// TIA Portal V17 export
// export: Created 2025-04-09T08:02:53.4997425Z, ExportSetting WithDefaults, DisplayName Totally Integrated Automation Portal, DisplayVersion V17 Update 8, DisplayName TIA Portal Openness, DisplayVersion V17 Update 8, DisplayName TIA Portal Version Control Interface, DisplayVersion V17, DisplayName SINAMICS Startdrive Advanced, DisplayVersion V17 SP2, DisplayName SINAMICS Startdrive G110M, G120, G120C, G120D, G120P, G115D, DisplayVersion V17 SP2, DisplayName SINAMICS Startdrive G130, G150, S120, S150, SINAMICS MV, S210, DisplayVersion V17 SP2, DisplayName STEP 7 Professional, DisplayVersion V17 Update 8, DisplayName SINUMERIK ONE STEP 7 Toolbox, DisplayVersion V17 Update 12, DisplayName SINUMERIK ONE PLC Basic Program Plus, DisplayVersion V17 Update 12, DisplayName SINUMERIK 840D sl STEP 7 Toolbox, DisplayVersion V17 Update 12, DisplayName STEP 7 Safety, DisplayVersion V17 Update 6, DisplayName WinCC Advanced, DisplayVersion V17 Update 8
FUNCTION "FC7000_SAFETY_DOORS" : Void   // FC7000, LAD
{ S7_Optimized_Access := 'FALSE' }
AUTHOR : ETXETAR
VERSION : 1.0
// stored: AutoNumber false, IsIECCheckEnabled false, SetENOAutomatically false, UDAEnableTagReadback false
BEGIN

REGION Network 1: CALL FC7002 UNIT 01 STATION 2 SAFETY DOOR
   // 2#0000_0001 OPTIONS 0 BIT 0 IMMEDIATE STOP REACTION OPTION
   // 2#0000_0010 OPTIONS 0 BIT 1 SEOC WARNING REACTION OPTION
   // 2#0000_0100 OPTIONS 0 BIT 2 CLOSED SENSOR INPUT OPTION
   // 2#0000_1000 OPTIONS 0 BIT 3 CIRCUIT E2 OPTION
   // 2#0001_0000 OPTIONS 0 BIT 4 PNEUMATIC DRIVE OPTION
   // 2#0010_0000 OPTIONS 0 BIT 5 GANTRY ROBOT OK TO OPEN OPTION
   // 2#0100_0000 OPTIONS 0 BIT 6 SPARE OPTION
   // 2#1000_0000 OPTIONS 0 BIT 7 SPARE OPTION
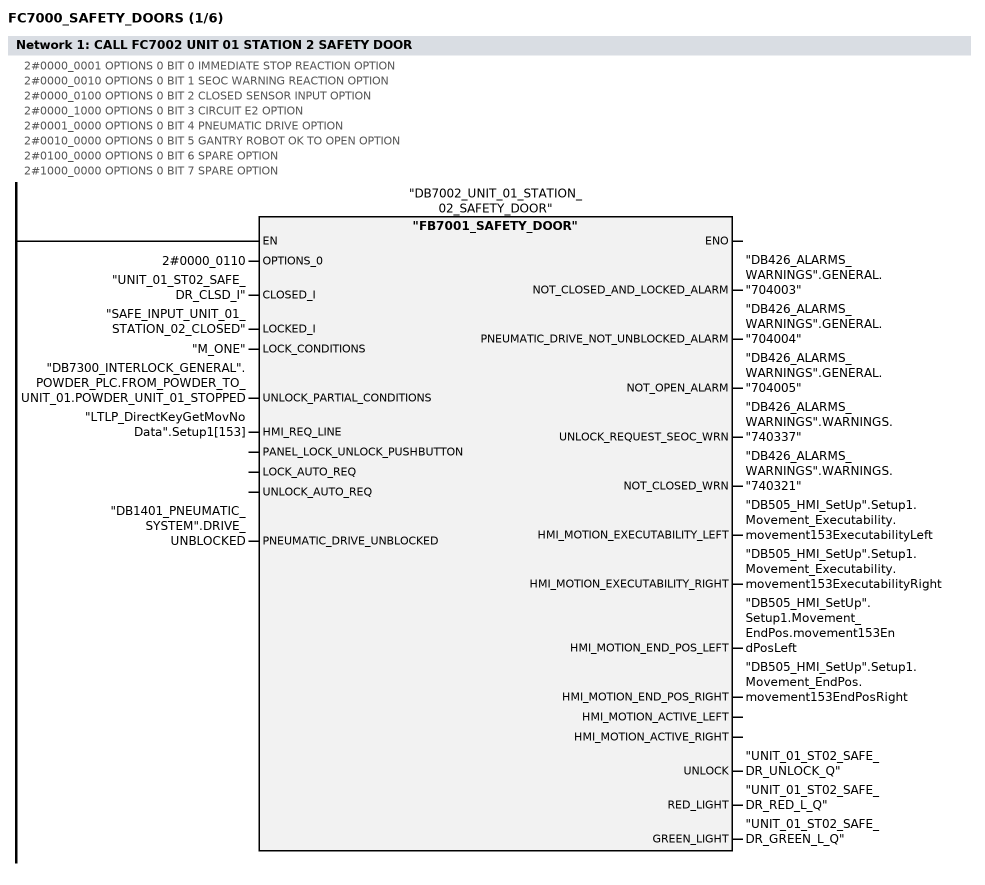
   RUNG wire#powerrail
      "DB7002_UNIT_01_STATION_02_SAFETY_DOOR"(OPTIONS_0 := 2#0000_0110, CLOSED_I := "UNIT_01_ST02_SAFE_DR_CLSD_I", LOCKED_I := "SAFE_INPUT_UNIT_01_STATION_02_CLOSED", LOCK_CONDITIONS := "M_ONE", UNLOCK_PARTIAL_CONDITIONS := "DB7300_INTERLOCK_GENERAL".POWDER_PLC.FROM_POWDER_TO_UNIT_01.POWDER_UNIT_01_STOPPED, HMI_REQ_LINE := "LTLP_DirectKeyGetMovNoData".Setup1[153], PANEL_LOCK_UNLOCK_PUSHBUTTON :=, LOCK_AUTO_REQ :=, UNLOCK_AUTO_REQ :=, PNEUMATIC_DRIVE_UNBLOCKED := "DB1401_PNEUMATIC_SYSTEM".DRIVE_UNBLOCKED, NOT_CLOSED_AND_LOCKED_ALARM => "DB426_ALARMS_WARNINGS".GENERAL."704003", PNEUMATIC_DRIVE_NOT_UNBLOCKED_ALARM => "DB426_ALARMS_WARNINGS".GENERAL."704004", NOT_OPEN_ALARM => "DB426_ALARMS_WARNINGS".GENERAL."704005", UNLOCK_REQUEST_SEOC_WRN => "DB426_ALARMS_WARNINGS".WARNINGS."740337", NOT_CLOSED_WRN => "DB426_ALARMS_WARNINGS".WARNINGS."740321", HMI_MOTION_EXECUTABILITY_LEFT => "DB505_HMI_SetUp".Setup1.Movement_Executability.movement153ExecutabilityLeft, HMI_MOTION_EXECUTABILITY_RIGHT => "DB505_HMI_SetUp".Setup1.Movement_Executability.movement153ExecutabilityRight, HMI_MOTION_END_POS_LEFT => "DB505_HMI_SetUp".Setup1.Movement_EndPos.movement153EndPosLeft, HMI_MOTION_END_POS_RIGHT => "DB505_HMI_SetUp".Setup1.Movement_EndPos.movement153EndPosRight, HMI_MOTION_ACTIVE_LEFT =>, HMI_MOTION_ACTIVE_RIGHT =>, UNLOCK => "UNIT_01_ST02_SAFE_DR_UNLOCK_Q", RED_LIGHT => "UNIT_01_ST02_SAFE_DR_RED_L_Q", GREEN_LIGHT => "UNIT_01_ST02_SAFE_DR_GREEN_L_Q")
   END_RUNG
   // the same network as SCL:
   "DB7002_UNIT_01_STATION_02_SAFETY_DOOR"(OPTIONS_0 := 2#0000_0110,   // "FB7001_SAFETY_DOOR"
                           CLOSED_I := "UNIT_01_ST02_SAFE_DR_CLSD_I",
                           LOCKED_I := "SAFE_INPUT_UNIT_01_STATION_02_CLOSED",
                           LOCK_CONDITIONS := "M_ONE",
                           UNLOCK_PARTIAL_CONDITIONS := "DB7300_INTERLOCK_GENERAL".POWDER_PLC.FROM_POWDER_TO_UNIT_01.POWDER_UNIT_01_STOPPED,
                           HMI_REQ_LINE := "LTLP_DirectKeyGetMovNoData".Setup1[153],
                           PNEUMATIC_DRIVE_UNBLOCKED := "DB1401_PNEUMATIC_SYSTEM".DRIVE_UNBLOCKED,
                           NOT_CLOSED_AND_LOCKED_ALARM => "DB426_ALARMS_WARNINGS".GENERAL."704003",
                           PNEUMATIC_DRIVE_NOT_UNBLOCKED_ALARM => "DB426_ALARMS_WARNINGS".GENERAL."704004",
                           NOT_OPEN_ALARM => "DB426_ALARMS_WARNINGS".GENERAL."704005",
                           UNLOCK_REQUEST_SEOC_WRN => "DB426_ALARMS_WARNINGS".WARNINGS."740337",
                           NOT_CLOSED_WRN => "DB426_ALARMS_WARNINGS".WARNINGS."740321",
                           HMI_MOTION_EXECUTABILITY_LEFT => "DB505_HMI_SetUp".Setup1.Movement_Executability.movement153ExecutabilityLeft,
                           HMI_MOTION_EXECUTABILITY_RIGHT => "DB505_HMI_SetUp".Setup1.Movement_Executability.movement153ExecutabilityRight,
                           HMI_MOTION_END_POS_LEFT => "DB505_HMI_SetUp".Setup1.Movement_EndPos.movement153EndPosLeft,
                           HMI_MOTION_END_POS_RIGHT => "DB505_HMI_SetUp".Setup1.Movement_EndPos.movement153EndPosRight,
                           UNLOCK => "UNIT_01_ST02_SAFE_DR_UNLOCK_Q",
                           RED_LIGHT => "UNIT_01_ST02_SAFE_DR_RED_L_Q",
                           GREEN_LIGHT => "UNIT_01_ST02_SAFE_DR_GREEN_L_Q");
END_REGION

REGION Network 2: CALL FC7002 UNIT 01 STATION 4 SAFETY DOOR
   // 2#0000_0001 OPTIONS 0 BIT 0 IMMEDIATE STOP REACTION OPTION
   // 2#0000_0010 OPTIONS 0 BIT 1 SEOC WARNING REACTION OPTION
   // 2#0000_0100 OPTIONS 0 BIT 2 CLOSED SENSOR INPUT OPTION
   // 2#0000_1000 OPTIONS 0 BIT 3 CIRCUIT E2 OPTION
   // 2#0001_0000 OPTIONS 0 BIT 4 PNEUMATIC DRIVE OPTION
   // 2#0010_0000 OPTIONS 0 BIT 5 GANTRY ROBOT OK TO OPEN OPTION
   // 2#0100_0000 OPTIONS 0 BIT 6 SPARE OPTION
   // 2#1000_0000 OPTIONS 0 BIT 7 SPARE OPTION
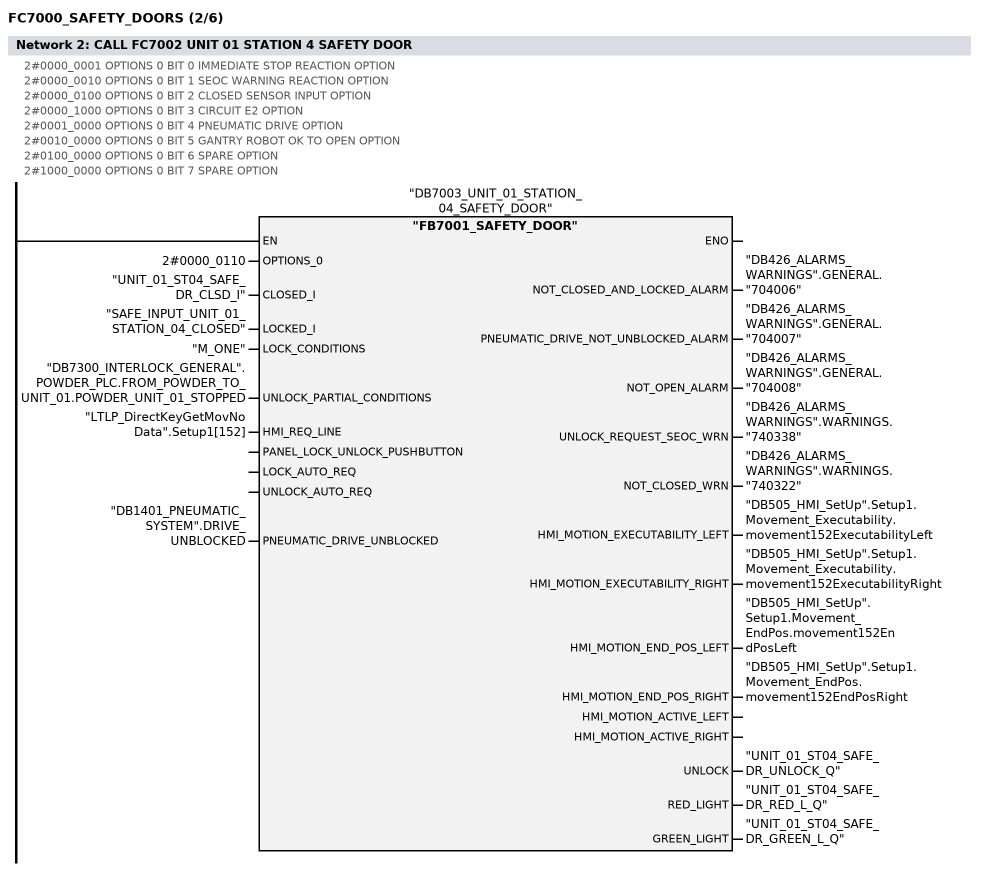
   RUNG wire#powerrail
      "DB7003_UNIT_01_STATION_04_SAFETY_DOOR"(OPTIONS_0 := 2#0000_0110, CLOSED_I := "UNIT_01_ST04_SAFE_DR_CLSD_I", LOCKED_I := "SAFE_INPUT_UNIT_01_STATION_04_CLOSED", LOCK_CONDITIONS := "M_ONE", UNLOCK_PARTIAL_CONDITIONS := "DB7300_INTERLOCK_GENERAL".POWDER_PLC.FROM_POWDER_TO_UNIT_01.POWDER_UNIT_01_STOPPED, HMI_REQ_LINE := "LTLP_DirectKeyGetMovNoData".Setup1[152], PANEL_LOCK_UNLOCK_PUSHBUTTON :=, LOCK_AUTO_REQ :=, UNLOCK_AUTO_REQ :=, PNEUMATIC_DRIVE_UNBLOCKED := "DB1401_PNEUMATIC_SYSTEM".DRIVE_UNBLOCKED, NOT_CLOSED_AND_LOCKED_ALARM => "DB426_ALARMS_WARNINGS".GENERAL."704006", PNEUMATIC_DRIVE_NOT_UNBLOCKED_ALARM => "DB426_ALARMS_WARNINGS".GENERAL."704007", NOT_OPEN_ALARM => "DB426_ALARMS_WARNINGS".GENERAL."704008", UNLOCK_REQUEST_SEOC_WRN => "DB426_ALARMS_WARNINGS".WARNINGS."740338", NOT_CLOSED_WRN => "DB426_ALARMS_WARNINGS".WARNINGS."740322", HMI_MOTION_EXECUTABILITY_LEFT => "DB505_HMI_SetUp".Setup1.Movement_Executability.movement152ExecutabilityLeft, HMI_MOTION_EXECUTABILITY_RIGHT => "DB505_HMI_SetUp".Setup1.Movement_Executability.movement152ExecutabilityRight, HMI_MOTION_END_POS_LEFT => "DB505_HMI_SetUp".Setup1.Movement_EndPos.movement152EndPosLeft, HMI_MOTION_END_POS_RIGHT => "DB505_HMI_SetUp".Setup1.Movement_EndPos.movement152EndPosRight, HMI_MOTION_ACTIVE_LEFT =>, HMI_MOTION_ACTIVE_RIGHT =>, UNLOCK => "UNIT_01_ST04_SAFE_DR_UNLOCK_Q", RED_LIGHT => "UNIT_01_ST04_SAFE_DR_RED_L_Q", GREEN_LIGHT => "UNIT_01_ST04_SAFE_DR_GREEN_L_Q")
   END_RUNG
   // the same network as SCL:
   "DB7003_UNIT_01_STATION_04_SAFETY_DOOR"(OPTIONS_0 := 2#0000_0110,   // "FB7001_SAFETY_DOOR"
                           CLOSED_I := "UNIT_01_ST04_SAFE_DR_CLSD_I",
                           LOCKED_I := "SAFE_INPUT_UNIT_01_STATION_04_CLOSED",
                           LOCK_CONDITIONS := "M_ONE",
                           UNLOCK_PARTIAL_CONDITIONS := "DB7300_INTERLOCK_GENERAL".POWDER_PLC.FROM_POWDER_TO_UNIT_01.POWDER_UNIT_01_STOPPED,
                           HMI_REQ_LINE := "LTLP_DirectKeyGetMovNoData".Setup1[152],
                           PNEUMATIC_DRIVE_UNBLOCKED := "DB1401_PNEUMATIC_SYSTEM".DRIVE_UNBLOCKED,
                           NOT_CLOSED_AND_LOCKED_ALARM => "DB426_ALARMS_WARNINGS".GENERAL."704006",
                           PNEUMATIC_DRIVE_NOT_UNBLOCKED_ALARM => "DB426_ALARMS_WARNINGS".GENERAL."704007",
                           NOT_OPEN_ALARM => "DB426_ALARMS_WARNINGS".GENERAL."704008",
                           UNLOCK_REQUEST_SEOC_WRN => "DB426_ALARMS_WARNINGS".WARNINGS."740338",
                           NOT_CLOSED_WRN => "DB426_ALARMS_WARNINGS".WARNINGS."740322",
                           HMI_MOTION_EXECUTABILITY_LEFT => "DB505_HMI_SetUp".Setup1.Movement_Executability.movement152ExecutabilityLeft,
                           HMI_MOTION_EXECUTABILITY_RIGHT => "DB505_HMI_SetUp".Setup1.Movement_Executability.movement152ExecutabilityRight,
                           HMI_MOTION_END_POS_LEFT => "DB505_HMI_SetUp".Setup1.Movement_EndPos.movement152EndPosLeft,
                           HMI_MOTION_END_POS_RIGHT => "DB505_HMI_SetUp".Setup1.Movement_EndPos.movement152EndPosRight,
                           UNLOCK => "UNIT_01_ST04_SAFE_DR_UNLOCK_Q",
                           RED_LIGHT => "UNIT_01_ST04_SAFE_DR_RED_L_Q",
                           GREEN_LIGHT => "UNIT_01_ST04_SAFE_DR_GREEN_L_Q");
END_REGION

REGION Network 3: CALL FC7001 UNIT 01 MAIN SAFETY DOOR
   // 2#0000_0001 OPTIONS 0 BIT 0 IMMEDIATE STOP REACTION OPTION
   // 2#0000_0010 OPTIONS 0 BIT 1 SEOC WARNING REACTION OPTION
   // 2#0000_0100 OPTIONS 0 BIT 2 CLOSED SENSOR INPUT OPTION
   // 2#0000_1000 OPTIONS 0 BIT 3 CIRCUIT E2 OPTION
   // 2#0001_0000 OPTIONS 0 BIT 4 PNEUMATIC DRIVE OPTION
   // 2#0010_0000 OPTIONS 0 BIT 5 GANTRY ROBOT OK TO OPEN OPTION
   // 2#0100_0000 OPTIONS 0 BIT 6 SPARE OPTION
   // 2#1000_0000 OPTIONS 0 BIT 7 SPARE OPTION
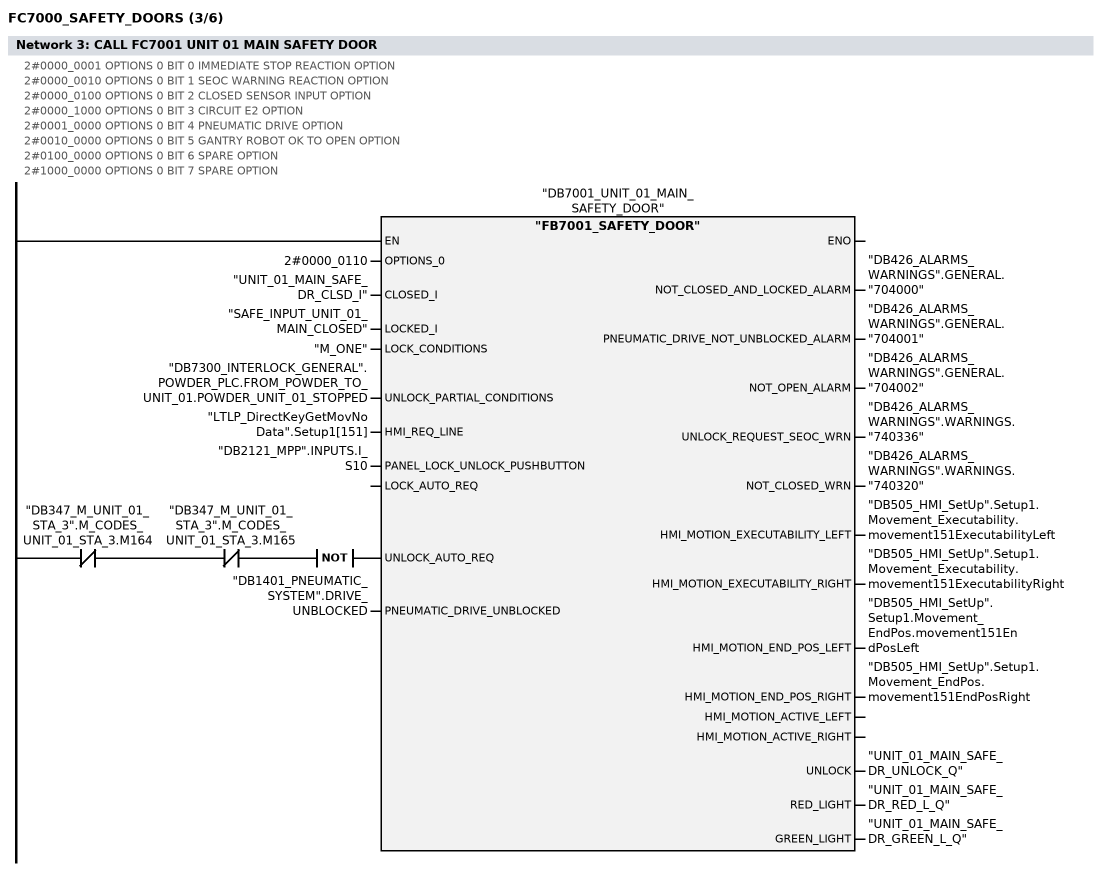
   RUNG wire#powerrail
      "DB7001_UNIT_01_MAIN_SAFETY_DOOR"(UNLOCK_AUTO_REQ := wire#w1, OPTIONS_0 := 2#0000_0110, CLOSED_I := "UNIT_01_MAIN_SAFE_DR_CLSD_I", LOCKED_I := "SAFE_INPUT_UNIT_01_MAIN_CLOSED", LOCK_CONDITIONS := "M_ONE", UNLOCK_PARTIAL_CONDITIONS := "DB7300_INTERLOCK_GENERAL".POWDER_PLC.FROM_POWDER_TO_UNIT_01.POWDER_UNIT_01_STOPPED, HMI_REQ_LINE := "LTLP_DirectKeyGetMovNoData".Setup1[151], PANEL_LOCK_UNLOCK_PUSHBUTTON := "DB2121_MPP".INPUTS.I_S10, LOCK_AUTO_REQ :=, PNEUMATIC_DRIVE_UNBLOCKED := "DB1401_PNEUMATIC_SYSTEM".DRIVE_UNBLOCKED, NOT_CLOSED_AND_LOCKED_ALARM => "DB426_ALARMS_WARNINGS".GENERAL."704000", PNEUMATIC_DRIVE_NOT_UNBLOCKED_ALARM => "DB426_ALARMS_WARNINGS".GENERAL."704001", NOT_OPEN_ALARM => "DB426_ALARMS_WARNINGS".GENERAL."704002", UNLOCK_REQUEST_SEOC_WRN => "DB426_ALARMS_WARNINGS".WARNINGS."740336", NOT_CLOSED_WRN => "DB426_ALARMS_WARNINGS".WARNINGS."740320", HMI_MOTION_EXECUTABILITY_LEFT => "DB505_HMI_SetUp".Setup1.Movement_Executability.movement151ExecutabilityLeft, HMI_MOTION_EXECUTABILITY_RIGHT => "DB505_HMI_SetUp".Setup1.Movement_Executability.movement151ExecutabilityRight, HMI_MOTION_END_POS_LEFT => "DB505_HMI_SetUp".Setup1.Movement_EndPos.movement151EndPosLeft, HMI_MOTION_END_POS_RIGHT => "DB505_HMI_SetUp".Setup1.Movement_EndPos.movement151EndPosRight, HMI_MOTION_ACTIVE_LEFT =>, HMI_MOTION_ACTIVE_RIGHT =>, UNLOCK => "UNIT_01_MAIN_SAFE_DR_UNLOCK_Q", RED_LIGHT => "UNIT_01_MAIN_SAFE_DR_RED_L_Q", GREEN_LIGHT => "UNIT_01_MAIN_SAFE_DR_GREEN_L_Q")
   END_RUNG
   RUNG wire#powerrail
      I_Contact( "DB347_M_UNIT_01_STA_3".M_CODES_UNIT_01_STA_3.M164 )
      I_Contact( "DB347_M_UNIT_01_STA_3".M_CODES_UNIT_01_STA_3.M165 )
      Not()
   END_RUNG wire#w1
   // the same network as SCL:
   "DB7001_UNIT_01_MAIN_SAFETY_DOOR"(OPTIONS_0 := 2#0000_0110,   // "FB7001_SAFETY_DOOR"
                           CLOSED_I := "UNIT_01_MAIN_SAFE_DR_CLSD_I",
                           LOCKED_I := "SAFE_INPUT_UNIT_01_MAIN_CLOSED",
                           LOCK_CONDITIONS := "M_ONE",
                           UNLOCK_PARTIAL_CONDITIONS := "DB7300_INTERLOCK_GENERAL".POWDER_PLC.FROM_POWDER_TO_UNIT_01.POWDER_UNIT_01_STOPPED,
                           HMI_REQ_LINE := "LTLP_DirectKeyGetMovNoData".Setup1[151],
                           PANEL_LOCK_UNLOCK_PUSHBUTTON := "DB2121_MPP".INPUTS.I_S10,
                           UNLOCK_AUTO_REQ := NOT (NOT "DB347_M_UNIT_01_STA_3".M_CODES_UNIT_01_STA_3.M164 AND NOT "DB347_M_UNIT_01_STA_3".M_CODES_UNIT_01_STA_3.M165),
                           PNEUMATIC_DRIVE_UNBLOCKED := "DB1401_PNEUMATIC_SYSTEM".DRIVE_UNBLOCKED,
                           NOT_CLOSED_AND_LOCKED_ALARM => "DB426_ALARMS_WARNINGS".GENERAL."704000",
                           PNEUMATIC_DRIVE_NOT_UNBLOCKED_ALARM => "DB426_ALARMS_WARNINGS".GENERAL."704001",
                           NOT_OPEN_ALARM => "DB426_ALARMS_WARNINGS".GENERAL."704002",
                           UNLOCK_REQUEST_SEOC_WRN => "DB426_ALARMS_WARNINGS".WARNINGS."740336",
                           NOT_CLOSED_WRN => "DB426_ALARMS_WARNINGS".WARNINGS."740320",
                           HMI_MOTION_EXECUTABILITY_LEFT => "DB505_HMI_SetUp".Setup1.Movement_Executability.movement151ExecutabilityLeft,
                           HMI_MOTION_EXECUTABILITY_RIGHT => "DB505_HMI_SetUp".Setup1.Movement_Executability.movement151ExecutabilityRight,
                           HMI_MOTION_END_POS_LEFT => "DB505_HMI_SetUp".Setup1.Movement_EndPos.movement151EndPosLeft,
                           HMI_MOTION_END_POS_RIGHT => "DB505_HMI_SetUp".Setup1.Movement_EndPos.movement151EndPosRight,
                           UNLOCK => "UNIT_01_MAIN_SAFE_DR_UNLOCK_Q",
                           RED_LIGHT => "UNIT_01_MAIN_SAFE_DR_RED_L_Q",
                           GREEN_LIGHT => "UNIT_01_MAIN_SAFE_DR_GREEN_L_Q");
END_REGION

REGION Network 4: CALL FC7012 UNIT 02 STATION 2 SAFETY DOOR
   // 2#0000_0001 OPTIONS 0 BIT 0 IMMEDIATE STOP REACTION OPTION
   // 2#0000_0010 OPTIONS 0 BIT 1 SEOC WARNING REACTION OPTION
   // 2#0000_0100 OPTIONS 0 BIT 2 CLOSED SENSOR INPUT OPTION
   // 2#0000_1000 OPTIONS 0 BIT 3 CIRCUIT E2 OPTION
   // 2#0001_0000 OPTIONS 0 BIT 4 PNEUMATIC DRIVE OPTION
   // 2#0010_0000 OPTIONS 0 BIT 5 GANTRY ROBOT OK TO OPEN OPTION
   // 2#0100_0000 OPTIONS 0 BIT 6 SPARE OPTION
   // 2#1000_0000 OPTIONS 0 BIT 7 SPARE OPTION
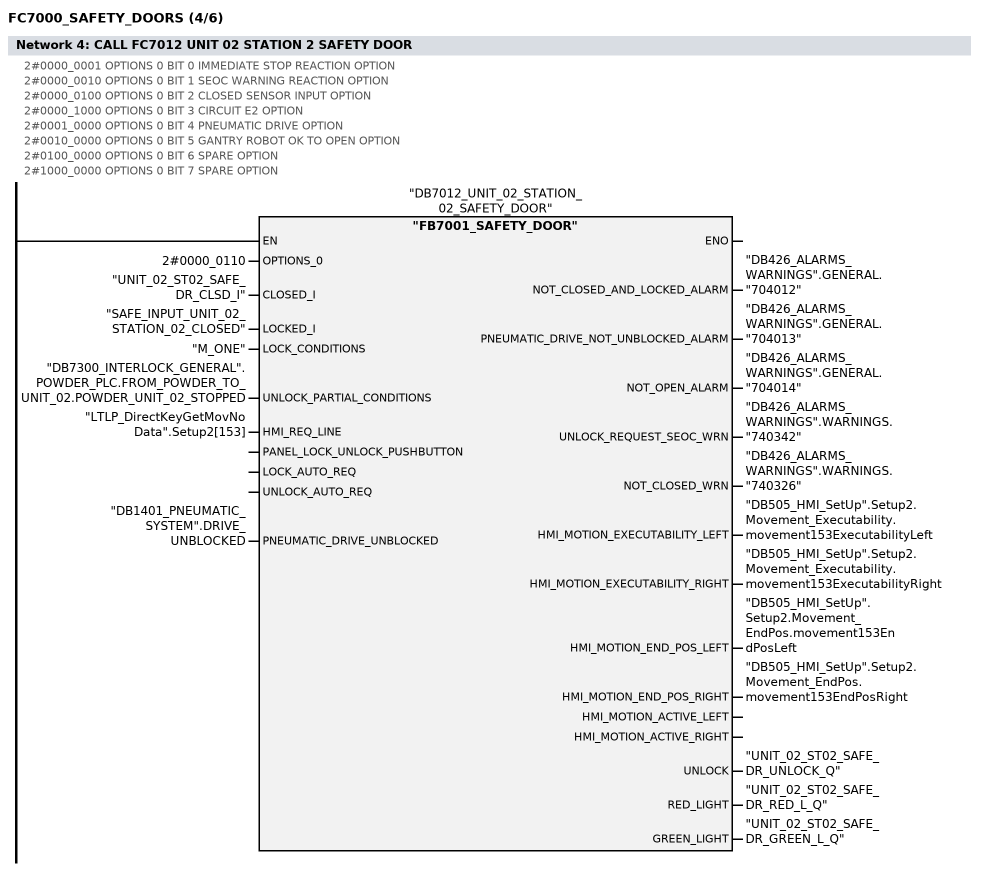
   RUNG wire#powerrail
      "DB7012_UNIT_02_STATION_02_SAFETY_DOOR"(OPTIONS_0 := 2#0000_0110, CLOSED_I := "UNIT_02_ST02_SAFE_DR_CLSD_I", LOCKED_I := "SAFE_INPUT_UNIT_02_STATION_02_CLOSED", LOCK_CONDITIONS := "M_ONE", UNLOCK_PARTIAL_CONDITIONS := "DB7300_INTERLOCK_GENERAL".POWDER_PLC.FROM_POWDER_TO_UNIT_02.POWDER_UNIT_02_STOPPED, HMI_REQ_LINE := "LTLP_DirectKeyGetMovNoData".Setup2[153], PANEL_LOCK_UNLOCK_PUSHBUTTON :=, LOCK_AUTO_REQ :=, UNLOCK_AUTO_REQ :=, PNEUMATIC_DRIVE_UNBLOCKED := "DB1401_PNEUMATIC_SYSTEM".DRIVE_UNBLOCKED, NOT_CLOSED_AND_LOCKED_ALARM => "DB426_ALARMS_WARNINGS".GENERAL."704012", PNEUMATIC_DRIVE_NOT_UNBLOCKED_ALARM => "DB426_ALARMS_WARNINGS".GENERAL."704013", NOT_OPEN_ALARM => "DB426_ALARMS_WARNINGS".GENERAL."704014", UNLOCK_REQUEST_SEOC_WRN => "DB426_ALARMS_WARNINGS".WARNINGS."740342", NOT_CLOSED_WRN => "DB426_ALARMS_WARNINGS".WARNINGS."740326", HMI_MOTION_EXECUTABILITY_LEFT => "DB505_HMI_SetUp".Setup2.Movement_Executability.movement153ExecutabilityLeft, HMI_MOTION_EXECUTABILITY_RIGHT => "DB505_HMI_SetUp".Setup2.Movement_Executability.movement153ExecutabilityRight, HMI_MOTION_END_POS_LEFT => "DB505_HMI_SetUp".Setup2.Movement_EndPos.movement153EndPosLeft, HMI_MOTION_END_POS_RIGHT => "DB505_HMI_SetUp".Setup2.Movement_EndPos.movement153EndPosRight, HMI_MOTION_ACTIVE_LEFT =>, HMI_MOTION_ACTIVE_RIGHT =>, UNLOCK => "UNIT_02_ST02_SAFE_DR_UNLOCK_Q", RED_LIGHT => "UNIT_02_ST02_SAFE_DR_RED_L_Q", GREEN_LIGHT => "UNIT_02_ST02_SAFE_DR_GREEN_L_Q")
   END_RUNG
   // the same network as SCL:
   "DB7012_UNIT_02_STATION_02_SAFETY_DOOR"(OPTIONS_0 := 2#0000_0110,   // "FB7001_SAFETY_DOOR"
                           CLOSED_I := "UNIT_02_ST02_SAFE_DR_CLSD_I",
                           LOCKED_I := "SAFE_INPUT_UNIT_02_STATION_02_CLOSED",
                           LOCK_CONDITIONS := "M_ONE",
                           UNLOCK_PARTIAL_CONDITIONS := "DB7300_INTERLOCK_GENERAL".POWDER_PLC.FROM_POWDER_TO_UNIT_02.POWDER_UNIT_02_STOPPED,
                           HMI_REQ_LINE := "LTLP_DirectKeyGetMovNoData".Setup2[153],
                           PNEUMATIC_DRIVE_UNBLOCKED := "DB1401_PNEUMATIC_SYSTEM".DRIVE_UNBLOCKED,
                           NOT_CLOSED_AND_LOCKED_ALARM => "DB426_ALARMS_WARNINGS".GENERAL."704012",
                           PNEUMATIC_DRIVE_NOT_UNBLOCKED_ALARM => "DB426_ALARMS_WARNINGS".GENERAL."704013",
                           NOT_OPEN_ALARM => "DB426_ALARMS_WARNINGS".GENERAL."704014",
                           UNLOCK_REQUEST_SEOC_WRN => "DB426_ALARMS_WARNINGS".WARNINGS."740342",
                           NOT_CLOSED_WRN => "DB426_ALARMS_WARNINGS".WARNINGS."740326",
                           HMI_MOTION_EXECUTABILITY_LEFT => "DB505_HMI_SetUp".Setup2.Movement_Executability.movement153ExecutabilityLeft,
                           HMI_MOTION_EXECUTABILITY_RIGHT => "DB505_HMI_SetUp".Setup2.Movement_Executability.movement153ExecutabilityRight,
                           HMI_MOTION_END_POS_LEFT => "DB505_HMI_SetUp".Setup2.Movement_EndPos.movement153EndPosLeft,
                           HMI_MOTION_END_POS_RIGHT => "DB505_HMI_SetUp".Setup2.Movement_EndPos.movement153EndPosRight,
                           UNLOCK => "UNIT_02_ST02_SAFE_DR_UNLOCK_Q",
                           RED_LIGHT => "UNIT_02_ST02_SAFE_DR_RED_L_Q",
                           GREEN_LIGHT => "UNIT_02_ST02_SAFE_DR_GREEN_L_Q");
END_REGION

REGION Network 5: CALL FC7013 UNIT 02 STATION 4 SAFETY DOOR
   // 2#0000_0001 OPTIONS 0 BIT 0 IMMEDIATE STOP REACTION OPTION
   // 2#0000_0010 OPTIONS 0 BIT 1 SEOC WARNING REACTION OPTION
   // 2#0000_0100 OPTIONS 0 BIT 2 CLOSED SENSOR INPUT OPTION
   // 2#0000_1000 OPTIONS 0 BIT 3 CIRCUIT E2 OPTION
   // 2#0001_0000 OPTIONS 0 BIT 4 PNEUMATIC DRIVE OPTION
   // 2#0010_0000 OPTIONS 0 BIT 5 GANTRY ROBOT OK TO OPEN OPTION
   // 2#0100_0000 OPTIONS 0 BIT 6 SPARE OPTION
   // 2#1000_0000 OPTIONS 0 BIT 7 SPARE OPTION
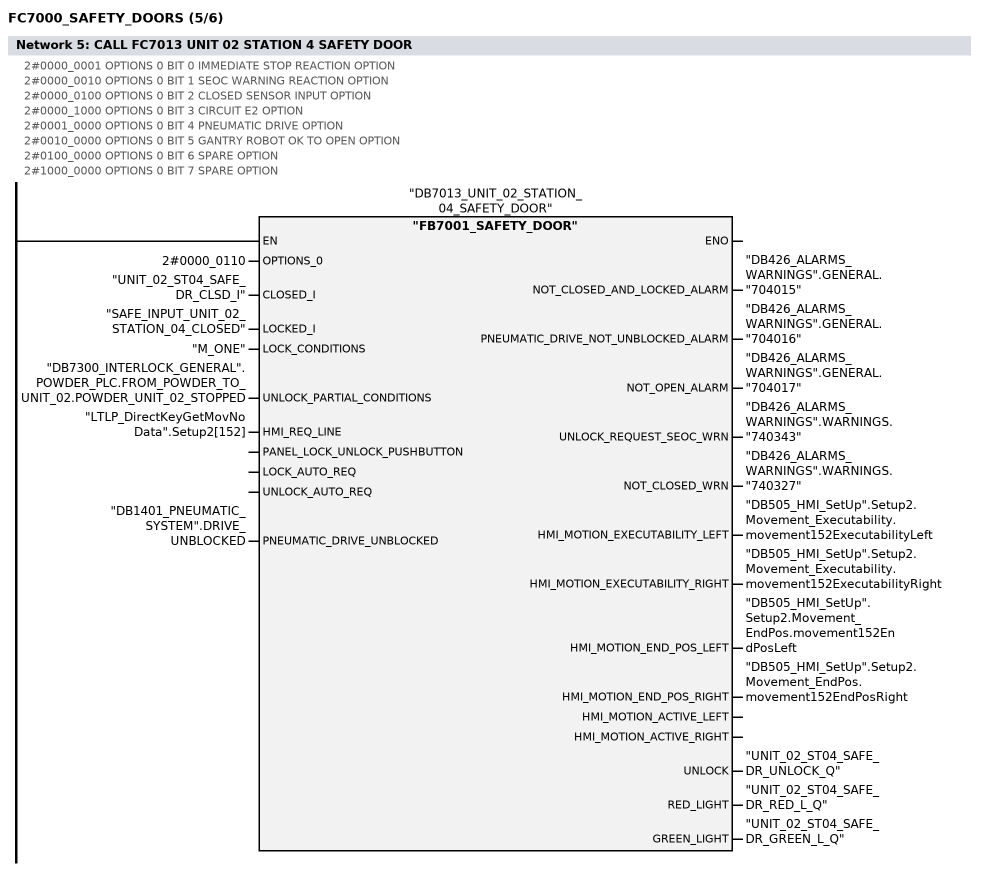
   RUNG wire#powerrail
      "DB7013_UNIT_02_STATION_04_SAFETY_DOOR"(OPTIONS_0 := 2#0000_0110, CLOSED_I := "UNIT_02_ST04_SAFE_DR_CLSD_I", LOCKED_I := "SAFE_INPUT_UNIT_02_STATION_04_CLOSED", LOCK_CONDITIONS := "M_ONE", UNLOCK_PARTIAL_CONDITIONS := "DB7300_INTERLOCK_GENERAL".POWDER_PLC.FROM_POWDER_TO_UNIT_02.POWDER_UNIT_02_STOPPED, HMI_REQ_LINE := "LTLP_DirectKeyGetMovNoData".Setup2[152], PANEL_LOCK_UNLOCK_PUSHBUTTON :=, LOCK_AUTO_REQ :=, UNLOCK_AUTO_REQ :=, PNEUMATIC_DRIVE_UNBLOCKED := "DB1401_PNEUMATIC_SYSTEM".DRIVE_UNBLOCKED, NOT_CLOSED_AND_LOCKED_ALARM => "DB426_ALARMS_WARNINGS".GENERAL."704015", PNEUMATIC_DRIVE_NOT_UNBLOCKED_ALARM => "DB426_ALARMS_WARNINGS".GENERAL."704016", NOT_OPEN_ALARM => "DB426_ALARMS_WARNINGS".GENERAL."704017", UNLOCK_REQUEST_SEOC_WRN => "DB426_ALARMS_WARNINGS".WARNINGS."740343", NOT_CLOSED_WRN => "DB426_ALARMS_WARNINGS".WARNINGS."740327", HMI_MOTION_EXECUTABILITY_LEFT => "DB505_HMI_SetUp".Setup2.Movement_Executability.movement152ExecutabilityLeft, HMI_MOTION_EXECUTABILITY_RIGHT => "DB505_HMI_SetUp".Setup2.Movement_Executability.movement152ExecutabilityRight, HMI_MOTION_END_POS_LEFT => "DB505_HMI_SetUp".Setup2.Movement_EndPos.movement152EndPosLeft, HMI_MOTION_END_POS_RIGHT => "DB505_HMI_SetUp".Setup2.Movement_EndPos.movement152EndPosRight, HMI_MOTION_ACTIVE_LEFT =>, HMI_MOTION_ACTIVE_RIGHT =>, UNLOCK => "UNIT_02_ST04_SAFE_DR_UNLOCK_Q", RED_LIGHT => "UNIT_02_ST04_SAFE_DR_RED_L_Q", GREEN_LIGHT => "UNIT_02_ST04_SAFE_DR_GREEN_L_Q")
   END_RUNG
   // the same network as SCL:
   "DB7013_UNIT_02_STATION_04_SAFETY_DOOR"(OPTIONS_0 := 2#0000_0110,   // "FB7001_SAFETY_DOOR"
                           CLOSED_I := "UNIT_02_ST04_SAFE_DR_CLSD_I",
                           LOCKED_I := "SAFE_INPUT_UNIT_02_STATION_04_CLOSED",
                           LOCK_CONDITIONS := "M_ONE",
                           UNLOCK_PARTIAL_CONDITIONS := "DB7300_INTERLOCK_GENERAL".POWDER_PLC.FROM_POWDER_TO_UNIT_02.POWDER_UNIT_02_STOPPED,
                           HMI_REQ_LINE := "LTLP_DirectKeyGetMovNoData".Setup2[152],
                           PNEUMATIC_DRIVE_UNBLOCKED := "DB1401_PNEUMATIC_SYSTEM".DRIVE_UNBLOCKED,
                           NOT_CLOSED_AND_LOCKED_ALARM => "DB426_ALARMS_WARNINGS".GENERAL."704015",
                           PNEUMATIC_DRIVE_NOT_UNBLOCKED_ALARM => "DB426_ALARMS_WARNINGS".GENERAL."704016",
                           NOT_OPEN_ALARM => "DB426_ALARMS_WARNINGS".GENERAL."704017",
                           UNLOCK_REQUEST_SEOC_WRN => "DB426_ALARMS_WARNINGS".WARNINGS."740343",
                           NOT_CLOSED_WRN => "DB426_ALARMS_WARNINGS".WARNINGS."740327",
                           HMI_MOTION_EXECUTABILITY_LEFT => "DB505_HMI_SetUp".Setup2.Movement_Executability.movement152ExecutabilityLeft,
                           HMI_MOTION_EXECUTABILITY_RIGHT => "DB505_HMI_SetUp".Setup2.Movement_Executability.movement152ExecutabilityRight,
                           HMI_MOTION_END_POS_LEFT => "DB505_HMI_SetUp".Setup2.Movement_EndPos.movement152EndPosLeft,
                           HMI_MOTION_END_POS_RIGHT => "DB505_HMI_SetUp".Setup2.Movement_EndPos.movement152EndPosRight,
                           UNLOCK => "UNIT_02_ST04_SAFE_DR_UNLOCK_Q",
                           RED_LIGHT => "UNIT_02_ST04_SAFE_DR_RED_L_Q",
                           GREEN_LIGHT => "UNIT_02_ST04_SAFE_DR_GREEN_L_Q");
END_REGION

REGION Network 6: CALL FC7011 UNIT 02 MAIN SAFETY DOOR
   // 2#0000_0001 OPTIONS 0 BIT 0 IMMEDIATE STOP REACTION OPTION
   // 2#0000_0010 OPTIONS 0 BIT 1 SEOC WARNING REACTION OPTION
   // 2#0000_0100 OPTIONS 0 BIT 2 CLOSED SENSOR INPUT OPTION
   // 2#0000_1000 OPTIONS 0 BIT 3 CIRCUIT E2 OPTION
   // 2#0001_0000 OPTIONS 0 BIT 4 PNEUMATIC DRIVE OPTION
   // 2#0010_0000 OPTIONS 0 BIT 5 GANTRY ROBOT OK TO OPEN OPTION
   // 2#0100_0000 OPTIONS 0 BIT 6 SPARE OPTION
   // 2#1000_0000 OPTIONS 0 BIT 7 SPARE OPTION
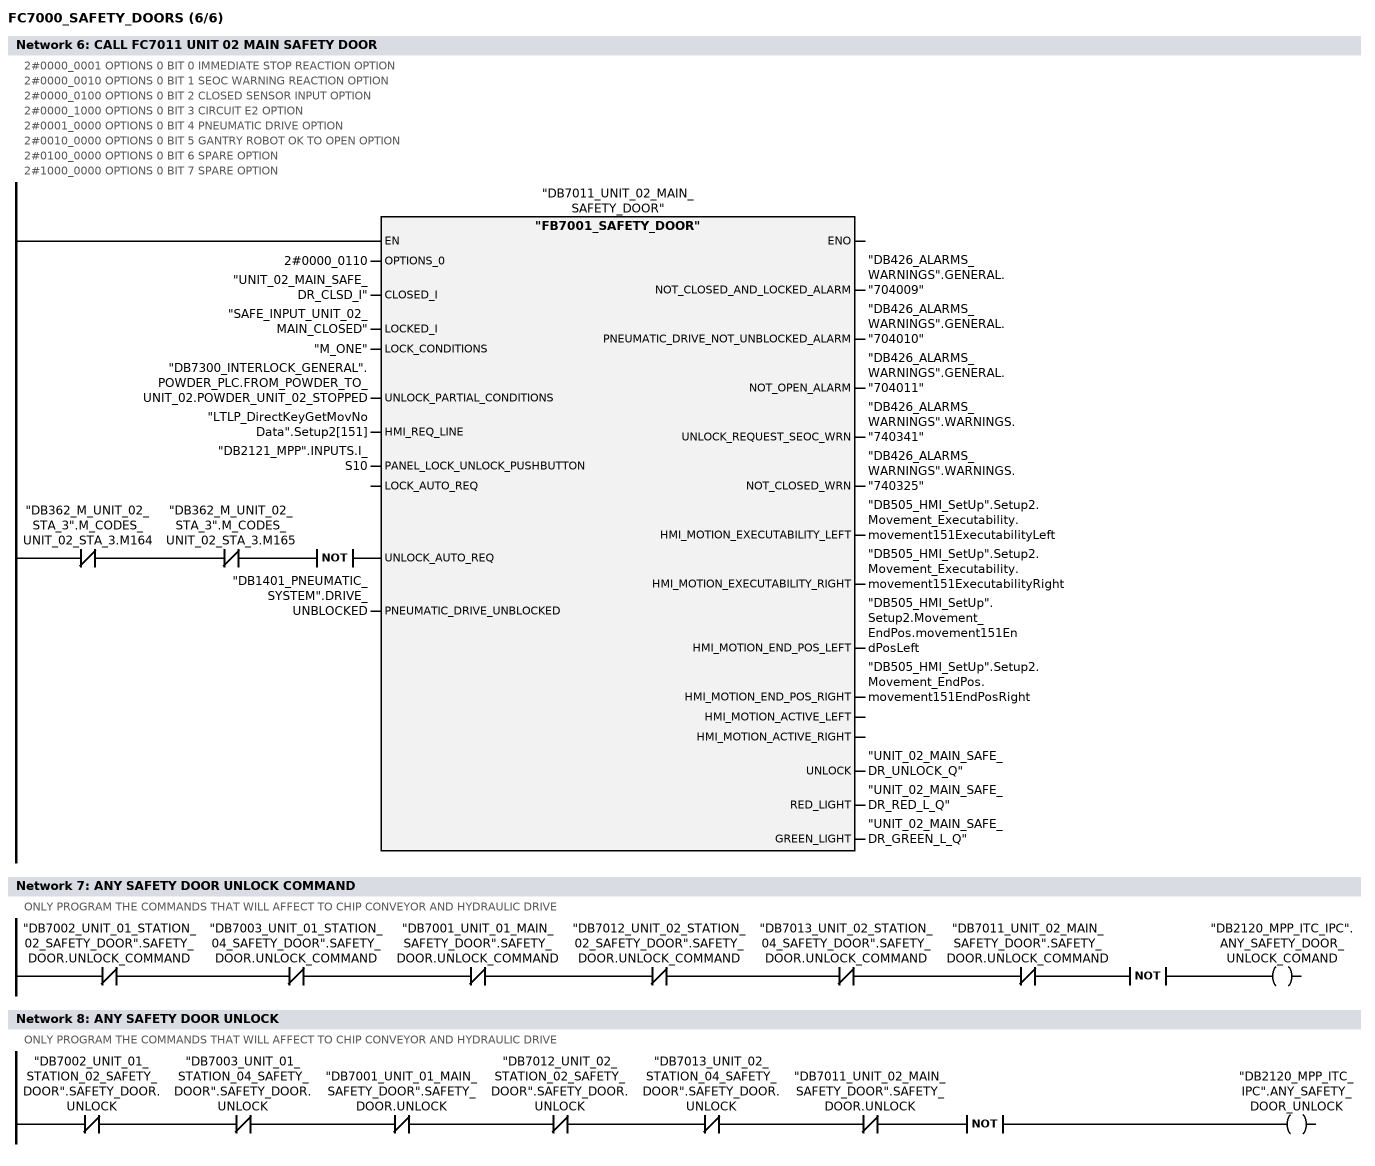
   RUNG wire#powerrail
      "DB7011_UNIT_02_MAIN_SAFETY_DOOR"(UNLOCK_AUTO_REQ := wire#w1, OPTIONS_0 := 2#0000_0110, CLOSED_I := "UNIT_02_MAIN_SAFE_DR_CLSD_I", LOCKED_I := "SAFE_INPUT_UNIT_02_MAIN_CLOSED", LOCK_CONDITIONS := "M_ONE", UNLOCK_PARTIAL_CONDITIONS := "DB7300_INTERLOCK_GENERAL".POWDER_PLC.FROM_POWDER_TO_UNIT_02.POWDER_UNIT_02_STOPPED, HMI_REQ_LINE := "LTLP_DirectKeyGetMovNoData".Setup2[151], PANEL_LOCK_UNLOCK_PUSHBUTTON := "DB2121_MPP".INPUTS.I_S10, LOCK_AUTO_REQ :=, PNEUMATIC_DRIVE_UNBLOCKED := "DB1401_PNEUMATIC_SYSTEM".DRIVE_UNBLOCKED, NOT_CLOSED_AND_LOCKED_ALARM => "DB426_ALARMS_WARNINGS".GENERAL."704009", PNEUMATIC_DRIVE_NOT_UNBLOCKED_ALARM => "DB426_ALARMS_WARNINGS".GENERAL."704010", NOT_OPEN_ALARM => "DB426_ALARMS_WARNINGS".GENERAL."704011", UNLOCK_REQUEST_SEOC_WRN => "DB426_ALARMS_WARNINGS".WARNINGS."740341", NOT_CLOSED_WRN => "DB426_ALARMS_WARNINGS".WARNINGS."740325", HMI_MOTION_EXECUTABILITY_LEFT => "DB505_HMI_SetUp".Setup2.Movement_Executability.movement151ExecutabilityLeft, HMI_MOTION_EXECUTABILITY_RIGHT => "DB505_HMI_SetUp".Setup2.Movement_Executability.movement151ExecutabilityRight, HMI_MOTION_END_POS_LEFT => "DB505_HMI_SetUp".Setup2.Movement_EndPos.movement151EndPosLeft, HMI_MOTION_END_POS_RIGHT => "DB505_HMI_SetUp".Setup2.Movement_EndPos.movement151EndPosRight, HMI_MOTION_ACTIVE_LEFT =>, HMI_MOTION_ACTIVE_RIGHT =>, UNLOCK => "UNIT_02_MAIN_SAFE_DR_UNLOCK_Q", RED_LIGHT => "UNIT_02_MAIN_SAFE_DR_RED_L_Q", GREEN_LIGHT => "UNIT_02_MAIN_SAFE_DR_GREEN_L_Q")
   END_RUNG
   RUNG wire#powerrail
      I_Contact( "DB362_M_UNIT_02_STA_3".M_CODES_UNIT_02_STA_3.M164 )
      I_Contact( "DB362_M_UNIT_02_STA_3".M_CODES_UNIT_02_STA_3.M165 )
      Not()
   END_RUNG wire#w1
   // the same network as SCL:
   "DB7011_UNIT_02_MAIN_SAFETY_DOOR"(OPTIONS_0 := 2#0000_0110,   // "FB7001_SAFETY_DOOR"
                           CLOSED_I := "UNIT_02_MAIN_SAFE_DR_CLSD_I",
                           LOCKED_I := "SAFE_INPUT_UNIT_02_MAIN_CLOSED",
                           LOCK_CONDITIONS := "M_ONE",
                           UNLOCK_PARTIAL_CONDITIONS := "DB7300_INTERLOCK_GENERAL".POWDER_PLC.FROM_POWDER_TO_UNIT_02.POWDER_UNIT_02_STOPPED,
                           HMI_REQ_LINE := "LTLP_DirectKeyGetMovNoData".Setup2[151],
                           PANEL_LOCK_UNLOCK_PUSHBUTTON := "DB2121_MPP".INPUTS.I_S10,
                           UNLOCK_AUTO_REQ := NOT (NOT "DB362_M_UNIT_02_STA_3".M_CODES_UNIT_02_STA_3.M164 AND NOT "DB362_M_UNIT_02_STA_3".M_CODES_UNIT_02_STA_3.M165),
                           PNEUMATIC_DRIVE_UNBLOCKED := "DB1401_PNEUMATIC_SYSTEM".DRIVE_UNBLOCKED,
                           NOT_CLOSED_AND_LOCKED_ALARM => "DB426_ALARMS_WARNINGS".GENERAL."704009",
                           PNEUMATIC_DRIVE_NOT_UNBLOCKED_ALARM => "DB426_ALARMS_WARNINGS".GENERAL."704010",
                           NOT_OPEN_ALARM => "DB426_ALARMS_WARNINGS".GENERAL."704011",
                           UNLOCK_REQUEST_SEOC_WRN => "DB426_ALARMS_WARNINGS".WARNINGS."740341",
                           NOT_CLOSED_WRN => "DB426_ALARMS_WARNINGS".WARNINGS."740325",
                           HMI_MOTION_EXECUTABILITY_LEFT => "DB505_HMI_SetUp".Setup2.Movement_Executability.movement151ExecutabilityLeft,
                           HMI_MOTION_EXECUTABILITY_RIGHT => "DB505_HMI_SetUp".Setup2.Movement_Executability.movement151ExecutabilityRight,
                           HMI_MOTION_END_POS_LEFT => "DB505_HMI_SetUp".Setup2.Movement_EndPos.movement151EndPosLeft,
                           HMI_MOTION_END_POS_RIGHT => "DB505_HMI_SetUp".Setup2.Movement_EndPos.movement151EndPosRight,
                           UNLOCK => "UNIT_02_MAIN_SAFE_DR_UNLOCK_Q",
                           RED_LIGHT => "UNIT_02_MAIN_SAFE_DR_RED_L_Q",
                           GREEN_LIGHT => "UNIT_02_MAIN_SAFE_DR_GREEN_L_Q");
END_REGION

REGION Network 7: ANY SAFETY DOOR UNLOCK COMMAND
   // ONLY PROGRAM THE COMMANDS THAT WILL AFFECT TO CHIP CONVEYOR AND HYDRAULIC DRIVE
   RUNG wire#powerrail
      I_Contact( "DB7002_UNIT_01_STATION_02_SAFETY_DOOR".SAFETY_DOOR.UNLOCK_COMMAND )
      I_Contact( "DB7003_UNIT_01_STATION_04_SAFETY_DOOR".SAFETY_DOOR.UNLOCK_COMMAND )
      I_Contact( "DB7001_UNIT_01_MAIN_SAFETY_DOOR".SAFETY_DOOR.UNLOCK_COMMAND )
      I_Contact( "DB7012_UNIT_02_STATION_02_SAFETY_DOOR".SAFETY_DOOR.UNLOCK_COMMAND )
      I_Contact( "DB7013_UNIT_02_STATION_04_SAFETY_DOOR".SAFETY_DOOR.UNLOCK_COMMAND )
      I_Contact( "DB7011_UNIT_02_MAIN_SAFETY_DOOR".SAFETY_DOOR.UNLOCK_COMMAND )
      Not()
      Coil( "DB2120_MPP_ITC_IPC".ANY_SAFETY_DOOR_UNLOCK_COMAND )
   END_RUNG
   // the same network as SCL:
   "DB2120_MPP_ITC_IPC".ANY_SAFETY_DOOR_UNLOCK_COMAND := NOT (NOT "DB7002_UNIT_01_STATION_02_SAFETY_DOOR".SAFETY_DOOR.UNLOCK_COMMAND AND NOT "DB7003_UNIT_01_STATION_04_SAFETY_DOOR".SAFETY_DOOR.UNLOCK_COMMAND AND NOT "DB7001_UNIT_01_MAIN_SAFETY_DOOR".SAFETY_DOOR.UNLOCK_COMMAND AND NOT "DB7012_UNIT_02_STATION_02_SAFETY_DOOR".SAFETY_DOOR.UNLOCK_COMMAND AND NOT "DB7013_UNIT_02_STATION_04_SAFETY_DOOR".SAFETY_DOOR.UNLOCK_COMMAND AND NOT "DB7011_UNIT_02_MAIN_SAFETY_DOOR".SAFETY_DOOR.UNLOCK_COMMAND);
END_REGION

REGION Network 8: ANY SAFETY DOOR UNLOCK
   // ONLY PROGRAM THE COMMANDS THAT WILL AFFECT TO CHIP CONVEYOR AND HYDRAULIC DRIVE
   RUNG wire#powerrail
      I_Contact( "DB7002_UNIT_01_STATION_02_SAFETY_DOOR".SAFETY_DOOR.UNLOCK )
      I_Contact( "DB7003_UNIT_01_STATION_04_SAFETY_DOOR".SAFETY_DOOR.UNLOCK )
      I_Contact( "DB7001_UNIT_01_MAIN_SAFETY_DOOR".SAFETY_DOOR.UNLOCK )
      I_Contact( "DB7012_UNIT_02_STATION_02_SAFETY_DOOR".SAFETY_DOOR.UNLOCK )
      I_Contact( "DB7013_UNIT_02_STATION_04_SAFETY_DOOR".SAFETY_DOOR.UNLOCK )
      I_Contact( "DB7011_UNIT_02_MAIN_SAFETY_DOOR".SAFETY_DOOR.UNLOCK )
      Not()
      Coil( "DB2120_MPP_ITC_IPC".ANY_SAFETY_DOOR_UNLOCK )
   END_RUNG
   // the same network as SCL:
   "DB2120_MPP_ITC_IPC".ANY_SAFETY_DOOR_UNLOCK := NOT (NOT "DB7002_UNIT_01_STATION_02_SAFETY_DOOR".SAFETY_DOOR.UNLOCK AND NOT "DB7003_UNIT_01_STATION_04_SAFETY_DOOR".SAFETY_DOOR.UNLOCK AND NOT "DB7001_UNIT_01_MAIN_SAFETY_DOOR".SAFETY_DOOR.UNLOCK AND NOT "DB7012_UNIT_02_STATION_02_SAFETY_DOOR".SAFETY_DOOR.UNLOCK AND NOT "DB7013_UNIT_02_STATION_04_SAFETY_DOOR".SAFETY_DOOR.UNLOCK AND NOT "DB7011_UNIT_02_MAIN_SAFETY_DOOR".SAFETY_DOOR.UNLOCK);
END_REGION
END_FUNCTION
